(* IEC 61131-3 sources: CodesysTest/alpha/export/FBs/FB_HMILight.pou, 3 files *)

(* ---- FB_HMILight.pou.st ---- *)
(*#-#-#-#-#-#-#-#-#-#---Declaration---#-#-#-#-#-#-#-#-#-#-#-#-#*)

FUNCTION_BLOCK FB_HMILight
VAR_INPUT
END_VAR
VAR_OUTPUT
	lightOutput : BOOL;
END_VAR
VAR
	_turnOn : BOOL;
	_blinkFast : BOOL;
	_blinkSlow : BOOL;
	blinker : OSCAT_BASIC.PWM_DC := (F := 1, DC := 0.5);
	slowBlinkSec : REAL := 1;
	fastBlinkSec : REAL := 0.5;
END_VAR
(*#-#-#-#-#-#-#-#-#-#---Implementation---#-#-#-#-#-#-#-#-#-#-#-#-#*)

IF _blinkFast THEN
	blinker.F := fastBlinkSec;
ELSIF _blinkSlow THEN
	blinker.F := slowBlinkSec;
END_IF

blinker(F:= , DC:= , Q=> );

lightOutput := _turnOn OR (blinker.Q AND (_blinkFast OR _blinkSlow));

(* ---- BlinkFast.m.st ---- *)
(*#-#-#-#-#-#-#-#-#-#---Declaration---#-#-#-#-#-#-#-#-#-#-#-#-#*)

METHOD BlinkFast
VAR_INPUT
END_VAR
(*#-#-#-#-#-#-#-#-#-#---Implementation---#-#-#-#-#-#-#-#-#-#-#-#-#*)

_blinkFast := TRUE;
_blinkSlow := FALSE;
_turnOn := FALSE;

(* ---- TurnOff.m.st ---- *)
(*#-#-#-#-#-#-#-#-#-#---Declaration---#-#-#-#-#-#-#-#-#-#-#-#-#*)

METHOD TurnOff
VAR_INPUT
END_VAR
(*#-#-#-#-#-#-#-#-#-#---Implementation---#-#-#-#-#-#-#-#-#-#-#-#-#*)

_blinkFast := FALSE;
_blinkSlow := FALSE;
_turnOn := FALSE;
